(* Logix 5000 project; controller GEA_Test_Chamber vendor 1 type 14 code 196 rev 32.14; software revision 32.04; part 8 of 11 *)
(* tags used below, declared in another part *)
   Heater_Cnt : COUNTER;
   LDO_Error_MSG : INT;
   LDO_LabView_Control : INT;
   LDO_LabView_Control2 : INT;
   LDO_Water_Outlet_Valve : REAL;
   LDO_Water_Outlet_Valve_Flow_SP : REAL;
   LDO_Water_Outlet_Valve_SP : REAL;
   Marcin : BOOL;
   Modbus_LabView_Data : raC_UDT_ModbusServerData;
   nLDO_Rate_REAL : REAL;
   Output_LDO : Output_LDO;

PROGRAM LDO_Chamber   (* main routine LDO_Main *)
VAR
   Act_Time : DINT[7] := ([0] := 2022, [1] := 8, [2] := 30, [4] := 36, [5] := 15, [6] := 396012);
   Actuators_OnOff_Heater : BOOL := 1;
   bPulse05Hz : BOOL := 1;
   bPulse0_1Hz : BOOL := 1;
   bPulse10Hz : BOOL;
   bPulse1Hz : BOOL;
   bPulse1min : BOOL;
   Counter : COUNTER[20] := ([0].PRE := 600, [1].PRE := 1200, [2].PRE := 3300, [3].PRE := 300, [4].PRE := 10, [5].PRE := 14100, [6].PRE := 300, [7].PRE := 2, [8].PRE := 14100, [9].PRE := 300, [10].PRE := 300, [11].PRE := 1500, [12].PRE := 180, [13].PRE := 1620, [14].PRE := 3300, [15].PRE := 300, [16].PRE := 1800, [17].PRE := 1800);
   DRK375_Flow_Change : BOOL;
   DRK375_Flow_InRange : BOOL := 1;
   DRK375_Temp_Change : BOOL;
   DRK375_Temp_InRange : BOOL := 1;
   Flow_Change_Step : INT;
   FVIR_Water_DRK375_Error : REAL := -175.0;
   GasSolenoidOnOff : BOOL := 1;
   Heater_OnOff : BOOL;
   LDO_DRK375_Start : BOOL;
   LDO_LabView_Comm_OK : BOOL;
   LDO_Oil_Step : INT;
   LDO_Step : INT;
   LDO_TestFlow : BOOL;
   LDO_Timer_Delay : TIMER[30] := ([0].PRE := 250, [20].PRE := 30000);
   LDO_Water_DRK375 : REAL := 50.0;
   LDO_Water_float : REAL := 9.0;
   LDO_Water_Flow_DRK375_REG : REAL := -175.0;
   LDO_Water_Flow_DRK375_SP : INT;
   LDO_Water_Outler_Flow : REAL;
   LDO_Water_Outlet : PID := (CTL := 41944064, CA := 1, PE := 1, DVNA := 1, SP := 135.0, KP := 1.0, KI := 0.1, MAXS := 4095.0, SO := 39.631687, MAXO := 50.0, MINO := 25.0, UPD := 0.1, PV := 134.7, ERR := -0.30000305, OUT := 39.631687, PVH := 200.0, DVP := 100.0, MAXI := 4095.0, MAXTIE := 4095.0, DATA[0] := 39.63901, DATA[1] := 52.630035, DATA[2] := 134.7, DATA[3] := -0.30000305, DATA[4] := 135.0, DATA[5] := 0.024420025, DATA[6] := 1.0, DATA[7] := 1.6, DATA[8] := 1.0, DATA[9] := 0.1, DATA[11] := 1.0, DATA[12] := 0.16666667, DATA[16] := 0.024420025);
   LDO_Water_Outlet_2 : PID := (CTL := -2139057280, EN := 1, PE := 1, INI := 1, OLH := 1, DVPA := 1, PVLA := 1, PVHA := 1, SP := 0.5803782, KP := 1.0, KI := 0.1, MAXS := 4095.0, SO := 100.0, MAXO := 100.0, UPD := 0.1, ERR := 0.5803782, OUT := 100.0, MAXI := 4095.0, MAXTIE := 4095.0, DATA[0] := 99.98566, DATA[3] := 0.5803782, DATA[4] := 0.5803782, DATA[5] := 0.024420025, DATA[6] := 1.0, DATA[7] := 1.6, DATA[8] := 1.0, DATA[9] := 0.1, DATA[11] := 1.0, DATA[12] := 0.16666667, DATA[16] := 0.024420025);
   LDO_Water_Outlet_HighLimit : REAL := 140.0;
   LDO_Water_Outlet_LowLimit : REAL := 130.0;
   LDO_Water_Outlet_Temp : REAL := 95.6;
   LDO_Water_Outlet_Valve_PID : REAL;
   LDO_Water_SP_float : REAL := 11.42;
   LDO_Water_Temp_DRK375_SP : INT;
   LDO_Water_Temp_float : REAL := 6.552;
   LDO_Water_Temp_SP_float : REAL := 7.552;
   LDO_WaterHeater_Step : INT := 70;
   Manual : Output_LDO;
   Max_Limit : REAL := 5.88;
   Min_limit : REAL := -4.12;
   New_Time : BOOL := 1;
   Oil_spray_08_ccmin : BOOL;
   Oil_spray_11_ccmin : BOOL;
   Oil_spray_133_ccmin : BOOL;
   ONS : BOOL[32] := ([0] := 1);
   PID_CV : REAL := 100.0;
   PID_puls : BOOL;
   puls_start : BOOL;
   puls_stop : BOOL;
   Pulse : BOOL[32] := ([10] := 1, [12] := 1, [20] := 1);
   Pulses : BOOL[32];
   Reset_Cnt : BOOL;
   Spare_Module : BOOL;
   Start_Test : BOOL;
   Start_Water_Flow : BOOL := 1;
   Step_10_Done : BOOL;
   Step_20_Done : BOOL;
   Step_25_Done : BOOL;
   Step_30_Done : BOOL;
   Step_40_Done : BOOL;
   Step_5_Done : BOOL;
   T_Diff_10 : DINT := 453959;
   T_Diff_20 : DINT := 453659;
   T_Diff_25 : DINT := 405359;
   T_Diff_30 : DINT := 403559;
   T_Diff_40 : DINT := 403379;
   T_Diff_5 : DINT := 455759;
   T_Diff_Step10 : T_DIFF := (T_Diff_sec := 453959);
   T_Diff_Step20 : T_DIFF := (T_Diff_sec := 453659);
   T_Diff_Step25 : T_DIFF := (T_Diff_sec := 405359);
   T_Diff_Step30 : T_DIFF := (T_Diff_sec := 403559);
   T_Diff_Step40 : T_DIFF := (T_Diff_sec := 403379);
   T_Diff_Step5 : T_DIFF := (T_Diff_sec := 455759);
   T_Diff_WaterStep10 : T_DIFF := (T_Diff_sec := 423359);
   T_Diff_WaterStep20 : T_DIFF := (T_Diff_sec := 420059);
   T_Diff_WaterStep40 : T_DIFF := (T_Diff_sec := 405359);
   T_Diff_WaterStep5 : T_DIFF;
   T_Diff_WaterStep50 : T_DIFF := (T_Diff_sec := 391259);
   T_Diff_WaterStep70 : T_DIFF := (T_Diff_sec := 2159);
   T_Diff_WaterStep80 : T_DIFF := (T_Diff_sec := 2459);
   Temp_cal_LDO : DINT := 2425;
   Temp_Change_Step : INT;
   test : BOOL;
   test_Heater_Ready : BOOL := 1;
   Time_Step_10 : DINT[7] := ([0] := 2022, [1] := 8, [2] := 24, [3] := 18, [4] := 30, [5] := 16, [6] := 35);
   Time_Step_20 : DINT[7] := ([0] := 2022, [1] := 8, [2] := 24, [3] := 18, [4] := 35, [5] := 16, [6] := 117);
   Time_Step_25 : DINT[7] := ([0] := 2022, [1] := 8, [2] := 25, [3] := 8, [5] := 16, [6] := 112);
   Time_Step_30 : DINT[7] := ([0] := 2022, [1] := 8, [2] := 25, [3] := 8, [4] := 30, [5] := 16, [6] := 92);
   Time_Step_40 : DINT[7] := ([0] := 2022, [1] := 8, [2] := 25, [3] := 8, [4] := 33, [5] := 16, [6] := 171);
   Time_Step_5 : DINT[7] := ([0] := 2022, [1] := 8, [2] := 24, [3] := 18, [5] := 16, [6] := 621647);
   Timer_Delay : TIMER[30] := ([0].PRE := 100, [0].ACC := 100, [0].EN := 1, [0].DN := 1, [1].PRE := 200, [2].PRE := 500, [3].PRE := 500);
   tof0_1sPulse : TIMER := (PRE := 100, ACC := 100);
   tof10sPulse : TIMER := (PRE := 10000, ACC := 8231, TT := 1, DN := 1);
   tof1sPulse : TIMER := (PRE := 500, ACC := 500);
   tof2sPulse : TIMER := (PRE := 2000, ACC := 236, TT := 1, DN := 1);
   tof30sPulse : TIMER := (PRE := 30000, ACC := 8241, TT := 1, DN := 1);
   ton0_1sPulse : TIMER := (PRE := 100, ACC := 36, EN := 1, TT := 1);
   ton10sPulse : TIMER := (PRE := 10000);
   ton1sPulse : TIMER := (PRE := 500, ACC := 231, EN := 1, TT := 1);
   ton2sPulse : TIMER := (PRE := 2000);
   ton30sPulse : TIMER := (PRE := 30000);
   TON_LifeBit_OFF : TIMER := (PRE := 10000);
   TON_LifeBit_ON : TIMER := (PRE := 10000, ACC := 10000, EN := 1, DN := 1);
   Water_Flow_Calc : REAL := 1084.1355;
   Water_Flow_Calc_float : REAL := 4677.2036;
   Water_Flow_DRK375 : INT := 4677;
   Water_Flow_DRK375_Last : INT := 19;
   Water_Outlet_Calc_LDO : DINT := 1937;
   Water_Outlet_InRange : BOOL;
   Water_Outlet_InRange_LDO : BOOL := 1;
   Water_Outlet_Temp_OK : BOOL;
   Water_Outlet_Valve_LDO : DINT;
   Water_Step_10 : DINT[7] := ([0] := 2022, [1] := 8, [2] := 25, [3] := 3, [5] := 16, [6] := 156);
   Water_Step_10_Done : BOOL;
   Water_Step_20 : DINT[7] := ([0] := 2022, [1] := 8, [2] := 25, [3] := 3, [4] := 55, [5] := 16, [6] := 196);
   Water_Step_20_Done : BOOL;
   Water_Step_40 : DINT;
   Water_Step_401 : DINT[7] := ([0] := 2022, [1] := 8, [2] := 25, [3] := 8, [5] := 16, [6] := 112);
   Water_Step_40_Done : BOOL;
   Water_Step_50 : DINT[7] := ([0] := 2022, [1] := 8, [2] := 25, [3] := 11, [4] := 55, [5] := 16, [6] := 229);
   Water_Step_50_Done : BOOL;
   Water_Step_70 : DINT[7] := ([0] := 2022, [1] := 8, [2] := 30, [5] := 16, [6] := 142);
   Water_Step_70_Done : BOOL;
   Water_Step_80 : DINT[7] := ([0] := 2022, [1] := 8, [2] := 29, [3] := 23, [4] := 55, [5] := 16, [6] := 90);
   Water_Step_80_Done : BOOL;
   Water_T_Diff_10 : DINT := 423359;
   Water_T_Diff_20 : DINT := 420059;
   Water_T_Diff_40 : DINT := 405359;
   Water_T_Diff_50 : DINT := 391259;
   Water_T_Diff_70 : DINT := 2159;
   Water_T_Diff_80 : DINT := 2459;
   Water_Temp_Calc : INT := 289;
   Water_Temp_Calc_float : REAL := 3093.016;
   Water_Temp_DRK375 : INT := 3093;
   Water_Temp_DRK375_Last : REAL := 70.0;
   Water_Time_Step_10 : DINT;
END_VAR

ROUTINE LDO_Control_Valve   (* ladder *)
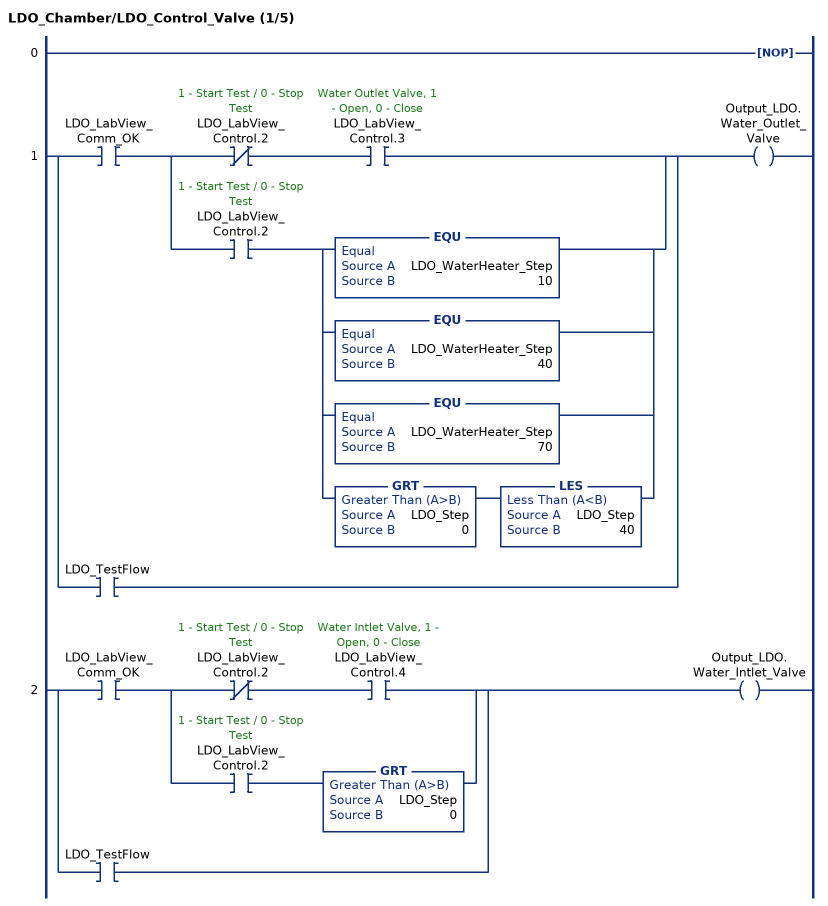
   0: NOP();
   1: [XIC(LDO_LabView_Comm_OK) [XIO(LDO_LabView_Control.2) XIC(LDO_LabView_Control.3) ,XIC(LDO_LabView_Control.2) [EQU(LDO_WaterHeater_Step,10) ,EQU(LDO_WaterHeater_Step,40) ,EQU(LDO_WaterHeater_Step,70) ,GRT(LDO_Step,0) LES(LDO_Step,40) ] ] ,XIC(LDO_TestFlow) ]OTE(Output_LDO.Water_Outlet_Valve);
   2: [XIC(LDO_LabView_Comm_OK) [XIO(LDO_LabView_Control.2) XIC(LDO_LabView_Control.4) ,XIC(LDO_LabView_Control.2) GRT(LDO_Step,0) ] ,XIC(LDO_TestFlow) ]OTE(Output_LDO.Water_Intlet_Valve);
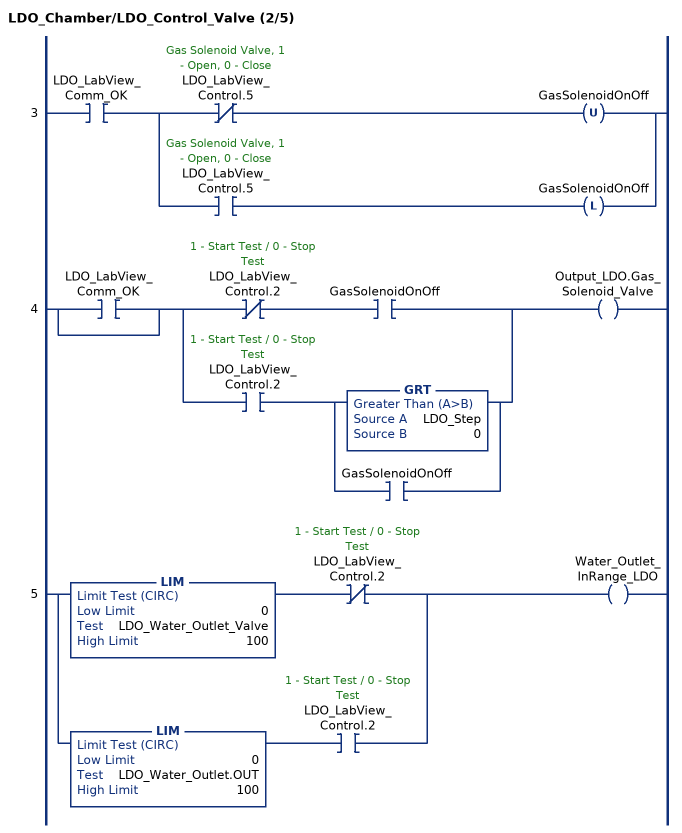
   3: XIC(LDO_LabView_Comm_OK)[XIO(LDO_LabView_Control.5) OTU(GasSolenoidOnOff) ,XIC(LDO_LabView_Control.5) OTL(GasSolenoidOnOff) ];
   4: [XIC(LDO_LabView_Comm_OK) ,][XIO(LDO_LabView_Control.2) XIC(GasSolenoidOnOff) ,XIC(LDO_LabView_Control.2) [GRT(LDO_Step,0) ,XIC(GasSolenoidOnOff) ] ]OTE(Output_LDO.Gas_Solenoid_Valve);
   5: [LIM(0,LDO_Water_Outlet_Valve,100) XIO(LDO_LabView_Control.2) ,LIM(0,LDO_Water_Outlet.OUT,100) XIC(LDO_LabView_Control.2) ]OTE(Water_Outlet_InRange_LDO);
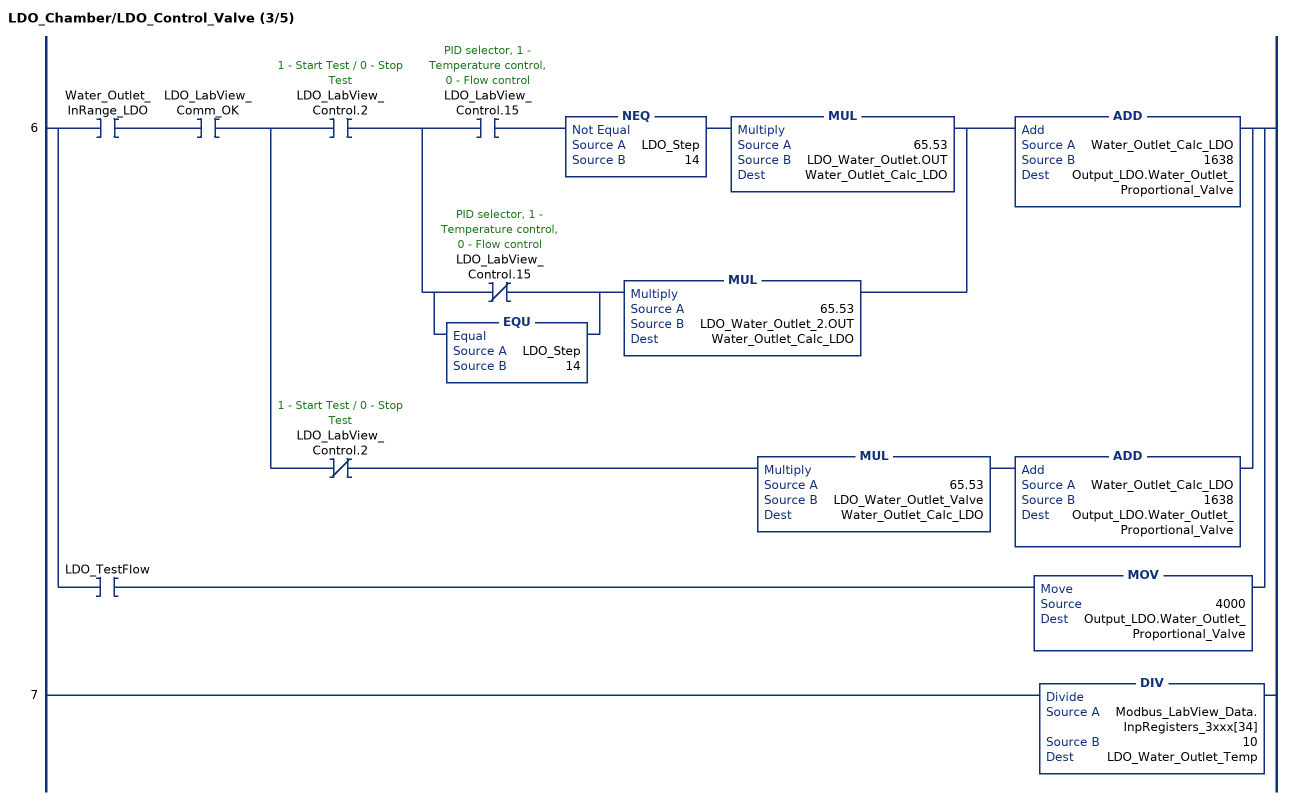
   6: [XIC(Water_Outlet_InRange_LDO) XIC(LDO_LabView_Comm_OK) [XIC(LDO_LabView_Control.2) [XIC(LDO_LabView_Control.15) NEQ(LDO_Step,14) MUL(65.53,LDO_Water_Outlet.OUT,Water_Outlet_Calc_LDO) ,[XIO(LDO_LabView_Control.15) ,EQU(LDO_Step,14) ] MUL(65.53,LDO_Water_Outlet_2.OUT,Water_Outlet_Calc_LDO) ] ADD(Water_Outlet_Calc_LDO,1638,Output_LDO.Water_Outlet_Proportional_Valve) ,XIO(LDO_LabView_Control.2) MUL(65.53,LDO_Water_Outlet_Valve,Water_Outlet_Calc_LDO) ADD(Water_Outlet_Calc_LDO,1638,Output_LDO.Water_Outlet_Proportional_Valve) ] ,XIC(LDO_TestFlow) MOV(4000,Output_LDO.Water_Outlet_Proportional_Valve) ];
   7: DIV(Modbus_LabView_Data.InpRegisters_3xxx[34],10,LDO_Water_Outlet_Temp);
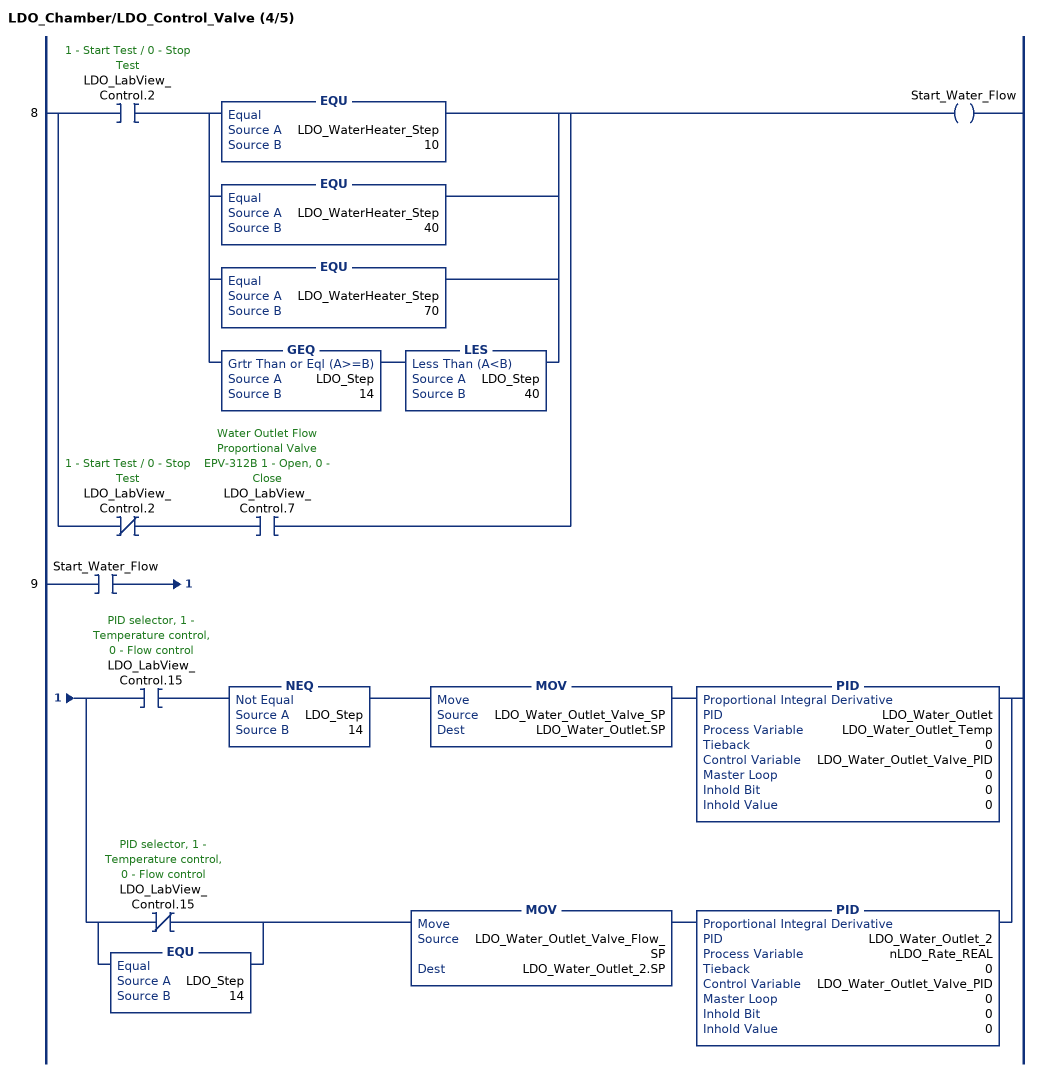
   8: [XIC(LDO_LabView_Control.2) [EQU(LDO_WaterHeater_Step,10) ,EQU(LDO_WaterHeater_Step,40) ,EQU(LDO_WaterHeater_Step,70) ,GEQ(LDO_Step,14) LES(LDO_Step,40) ] ,XIO(LDO_LabView_Control.2) XIC(LDO_LabView_Control.7) ]OTE(Start_Water_Flow);
   9: XIC(Start_Water_Flow)[XIC(LDO_LabView_Control.15) NEQ(LDO_Step,14) MOV(LDO_Water_Outlet_Valve_SP,LDO_Water_Outlet.SP) PID(LDO_Water_Outlet,LDO_Water_Outlet_Temp,0,LDO_Water_Outlet_Valve_PID,0,0,0) ,[XIO(LDO_LabView_Control.15) ,EQU(LDO_Step,14) ] MOV(LDO_Water_Outlet_Valve_Flow_SP,LDO_Water_Outlet_2.SP) PID(LDO_Water_Outlet_2,nLDO_Rate_REAL,0,LDO_Water_Outlet_Valve_PID,0,0,0) ];
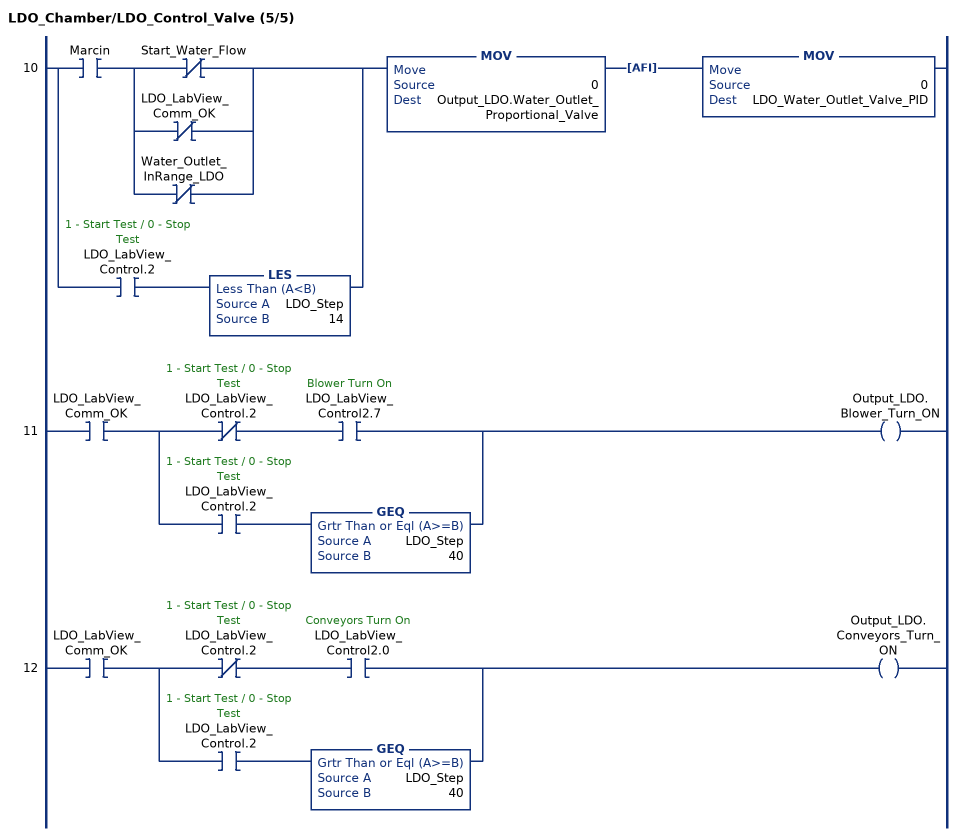
   10: [XIC(Marcin) [XIO(Start_Water_Flow) ,XIO(LDO_LabView_Comm_OK) ,XIO(Water_Outlet_InRange_LDO) ] ,XIC(LDO_LabView_Control.2) LES(LDO_Step,14) ]MOV(0,Output_LDO.Water_Outlet_Proportional_Valve)AFI()MOV(0,LDO_Water_Outlet_Valve_PID);
   11: XIC(LDO_LabView_Comm_OK)[XIO(LDO_LabView_Control.2) XIC(LDO_LabView_Control2.7) ,XIC(LDO_LabView_Control.2) GEQ(LDO_Step,40) ]OTE(Output_LDO.Blower_Turn_ON);
   12: XIC(LDO_LabView_Comm_OK)[XIO(LDO_LabView_Control.2) XIC(LDO_LabView_Control2.0) ,XIC(LDO_LabView_Control.2) GEQ(LDO_Step,40) ]OTE(Output_LDO.Conveyors_Turn_ON);
END_ROUTINE

ROUTINE LDO_Error_MSG   (* ladder *)
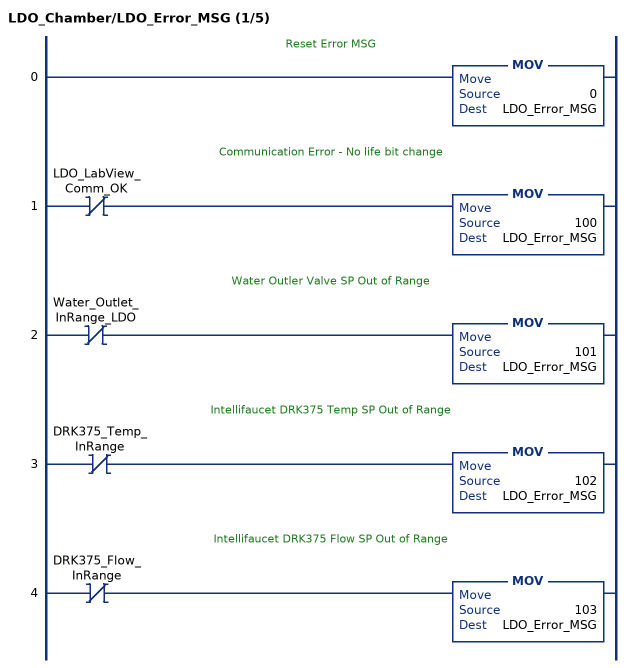
   // Reset Error MSG
   0: MOV(0,LDO_Error_MSG);
   // Communication Error - No life bit change
   1: XIO(LDO_LabView_Comm_OK)MOV(100,LDO_Error_MSG);
   // Water Outler Valve SP Out of Range
   2: XIO(Water_Outlet_InRange_LDO)MOV(101,LDO_Error_MSG);
   // Intellifaucet DRK375 Temp SP Out of Range
   3: XIO(DRK375_Temp_InRange)MOV(102,LDO_Error_MSG);
   // Intellifaucet DRK375 Flow SP Out of Range
   4: XIO(DRK375_Flow_InRange)MOV(103,LDO_Error_MSG);
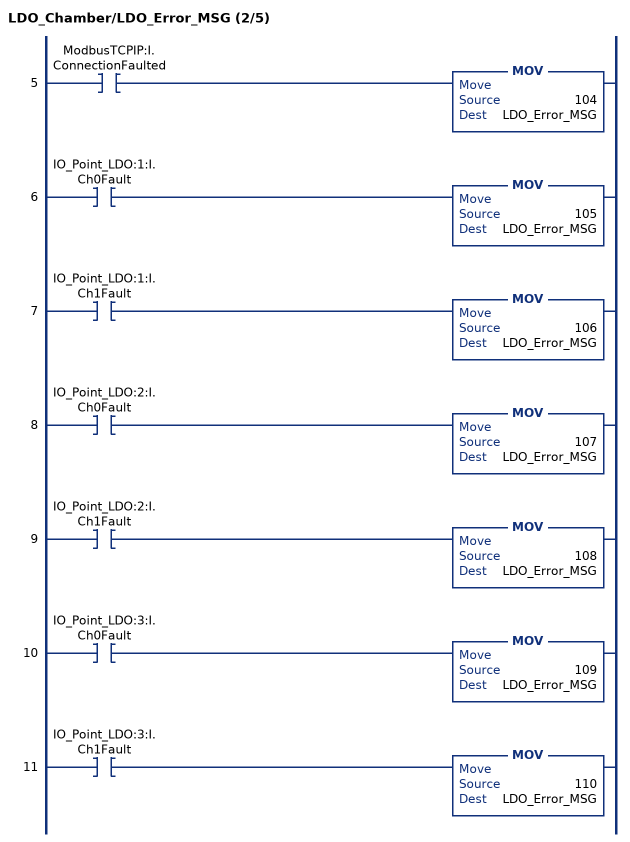
   5: XIC(ModbusTCPIP:I.ConnectionFaulted)MOV(104,LDO_Error_MSG);
   6: XIC(IO_Point_LDO:1:I.Ch0Fault)MOV(105,LDO_Error_MSG);
   7: XIC(IO_Point_LDO:1:I.Ch1Fault)MOV(106,LDO_Error_MSG);
   8: XIC(IO_Point_LDO:2:I.Ch0Fault)MOV(107,LDO_Error_MSG);
   9: XIC(IO_Point_LDO:2:I.Ch1Fault)MOV(108,LDO_Error_MSG);
   10: XIC(IO_Point_LDO:3:I.Ch0Fault)MOV(109,LDO_Error_MSG);
   11: XIC(IO_Point_LDO:3:I.Ch1Fault)MOV(110,LDO_Error_MSG);
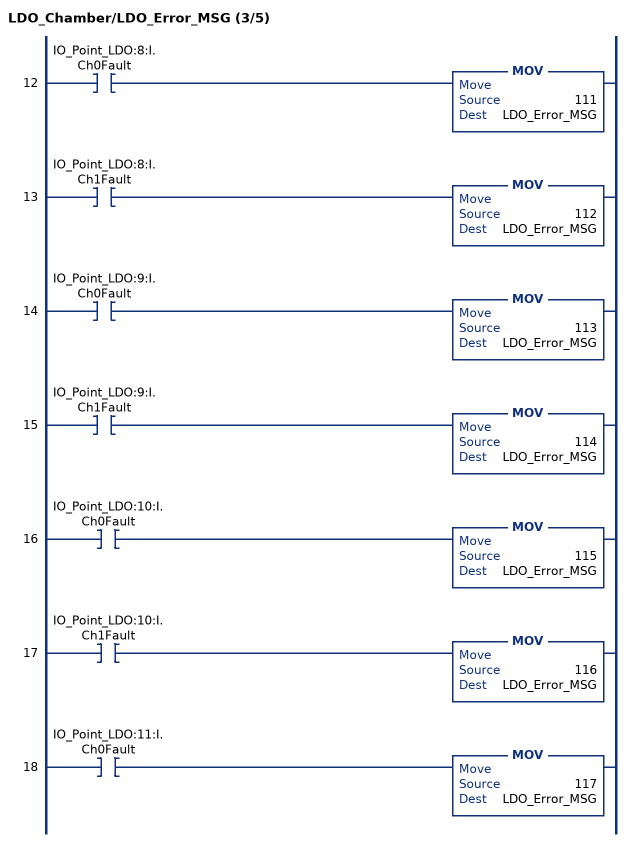
   12: XIC(IO_Point_LDO:8:I.Ch0Fault)MOV(111,LDO_Error_MSG);
   13: XIC(IO_Point_LDO:8:I.Ch1Fault)MOV(112,LDO_Error_MSG);
   14: XIC(IO_Point_LDO:9:I.Ch0Fault)MOV(113,LDO_Error_MSG);
   15: XIC(IO_Point_LDO:9:I.Ch1Fault)MOV(114,LDO_Error_MSG);
   16: XIC(IO_Point_LDO:10:I.Ch0Fault)MOV(115,LDO_Error_MSG);
   17: XIC(IO_Point_LDO:10:I.Ch1Fault)MOV(116,LDO_Error_MSG);
   18: XIC(IO_Point_LDO:11:I.Ch0Fault)MOV(117,LDO_Error_MSG);
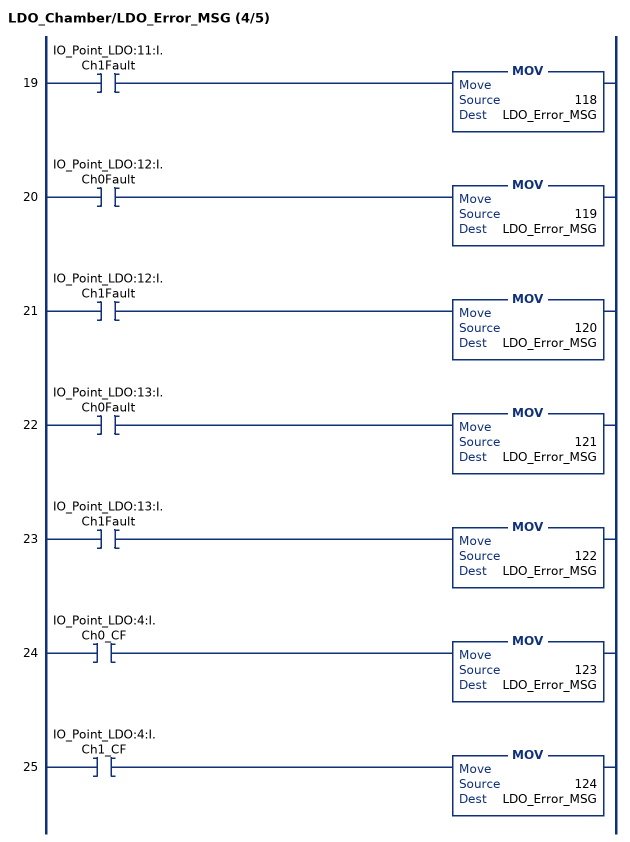
   19: XIC(IO_Point_LDO:11:I.Ch1Fault)MOV(118,LDO_Error_MSG);
   20: XIC(IO_Point_LDO:12:I.Ch0Fault)MOV(119,LDO_Error_MSG);
   21: XIC(IO_Point_LDO:12:I.Ch1Fault)MOV(120,LDO_Error_MSG);
   22: XIC(IO_Point_LDO:13:I.Ch0Fault)MOV(121,LDO_Error_MSG);
   23: XIC(IO_Point_LDO:13:I.Ch1Fault)MOV(122,LDO_Error_MSG);
   24: XIC(IO_Point_LDO:4:I.Ch0_CF)MOV(123,LDO_Error_MSG);
   25: XIC(IO_Point_LDO:4:I.Ch1_CF)MOV(124,LDO_Error_MSG);
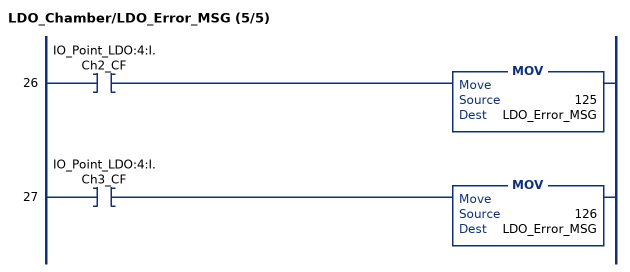
   26: XIC(IO_Point_LDO:4:I.Ch2_CF)MOV(125,LDO_Error_MSG);
   27: XIC(IO_Point_LDO:4:I.Ch3_CF)MOV(126,LDO_Error_MSG);
END_ROUTINE

ROUTINE LDO_Heater_OnOff   (* ladder *)
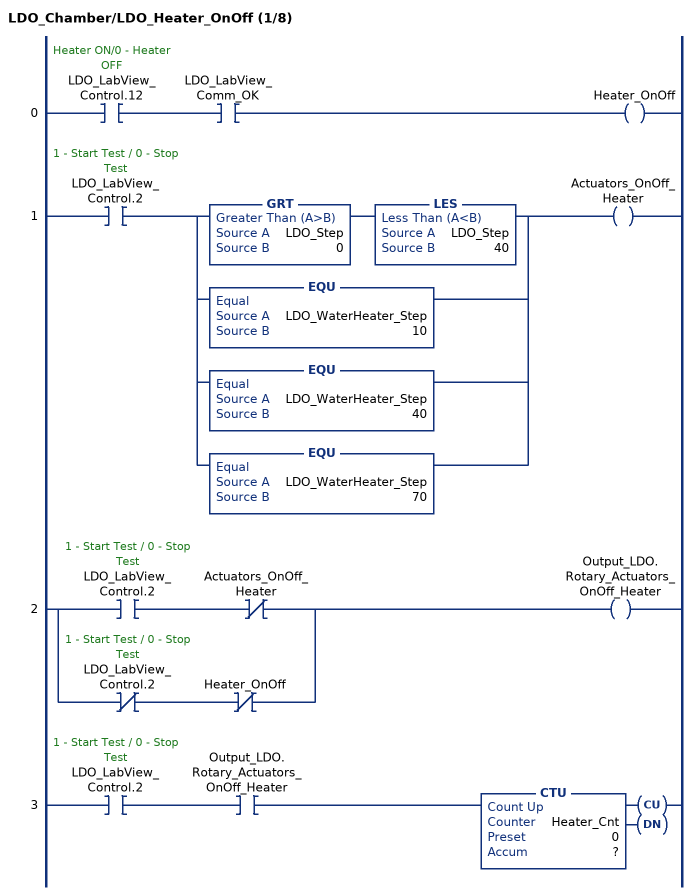
   0: XIC(LDO_LabView_Control.12)XIC(LDO_LabView_Comm_OK)OTE(Heater_OnOff);
   1: XIC(LDO_LabView_Control.2)[GRT(LDO_Step,0) LES(LDO_Step,40) ,EQU(LDO_WaterHeater_Step,10) ,EQU(LDO_WaterHeater_Step,40) ,EQU(LDO_WaterHeater_Step,70) ]OTE(Actuators_OnOff_Heater);
   2: [XIC(LDO_LabView_Control.2) XIO(Actuators_OnOff_Heater) ,XIO(LDO_LabView_Control.2) XIO(Heater_OnOff) ]OTE(Output_LDO.Rotary_Actuators_OnOff_Heater);
   3: XIC(LDO_LabView_Control.2)XIC(Output_LDO.Rotary_Actuators_OnOff_Heater)CTU(Heater_Cnt,?,?);
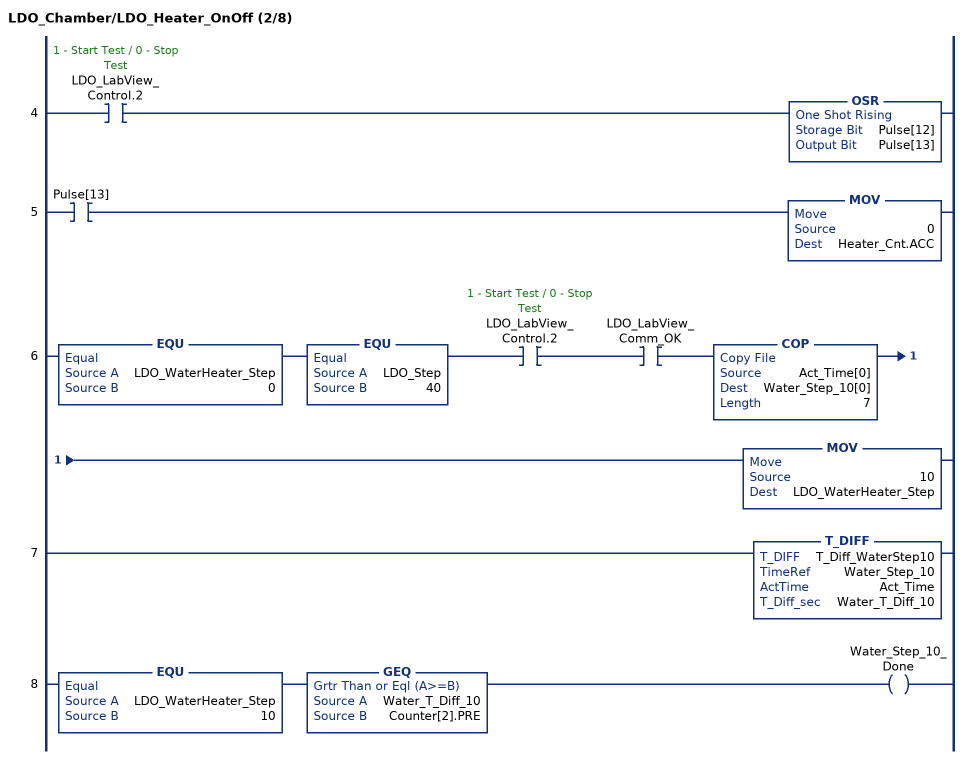
   4: XIC(LDO_LabView_Control.2)OSR(Pulse[12],Pulse[13]);
   5: XIC(Pulse[13])MOV(0,Heater_Cnt.ACC);
   6: EQU(LDO_WaterHeater_Step,0)EQU(LDO_Step,40)XIC(LDO_LabView_Control.2)XIC(LDO_LabView_Comm_OK)COP(Act_Time[0],Water_Step_10[0],7)MOV(10,LDO_WaterHeater_Step);
   7: T_DIFF(T_Diff_WaterStep10,Water_Step_10,Act_Time,Water_T_Diff_10);
   8: EQU(LDO_WaterHeater_Step,10)GEQ(Water_T_Diff_10,Counter[2].PRE)OTE(Water_Step_10_Done);
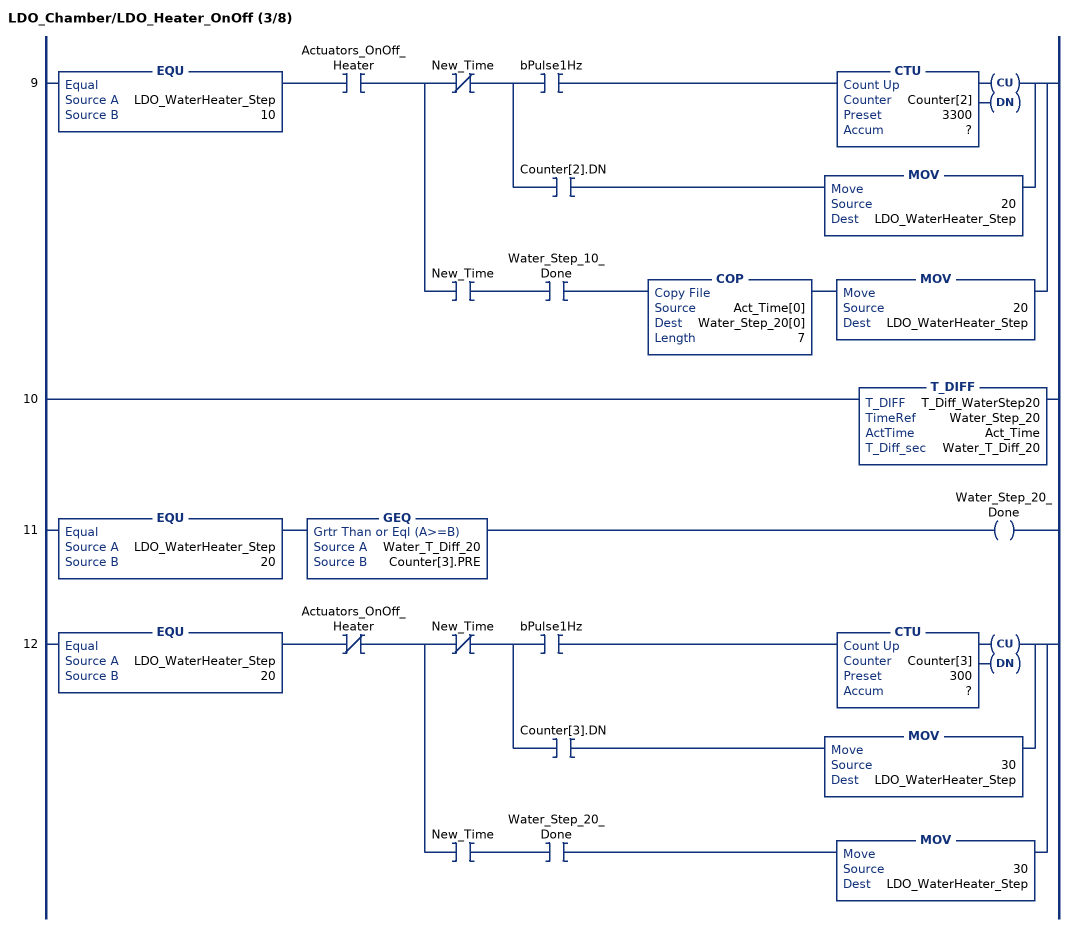
   9: EQU(LDO_WaterHeater_Step,10)XIC(Actuators_OnOff_Heater)[XIO(New_Time) [XIC(bPulse1Hz) CTU(Counter[2],?,?) ,XIC(Counter[2].DN) MOV(20,LDO_WaterHeater_Step) ] ,XIC(New_Time) XIC(Water_Step_10_Done) COP(Act_Time[0],Water_Step_20[0],7) MOV(20,LDO_WaterHeater_Step) ];
   10: T_DIFF(T_Diff_WaterStep20,Water_Step_20,Act_Time,Water_T_Diff_20);
   11: EQU(LDO_WaterHeater_Step,20)GEQ(Water_T_Diff_20,Counter[3].PRE)OTE(Water_Step_20_Done);
   12: EQU(LDO_WaterHeater_Step,20)XIO(Actuators_OnOff_Heater)[XIO(New_Time) [XIC(bPulse1Hz) CTU(Counter[3],?,?) ,XIC(Counter[3].DN) MOV(30,LDO_WaterHeater_Step) ] ,XIC(New_Time) XIC(Water_Step_20_Done) MOV(30,LDO_WaterHeater_Step) ];
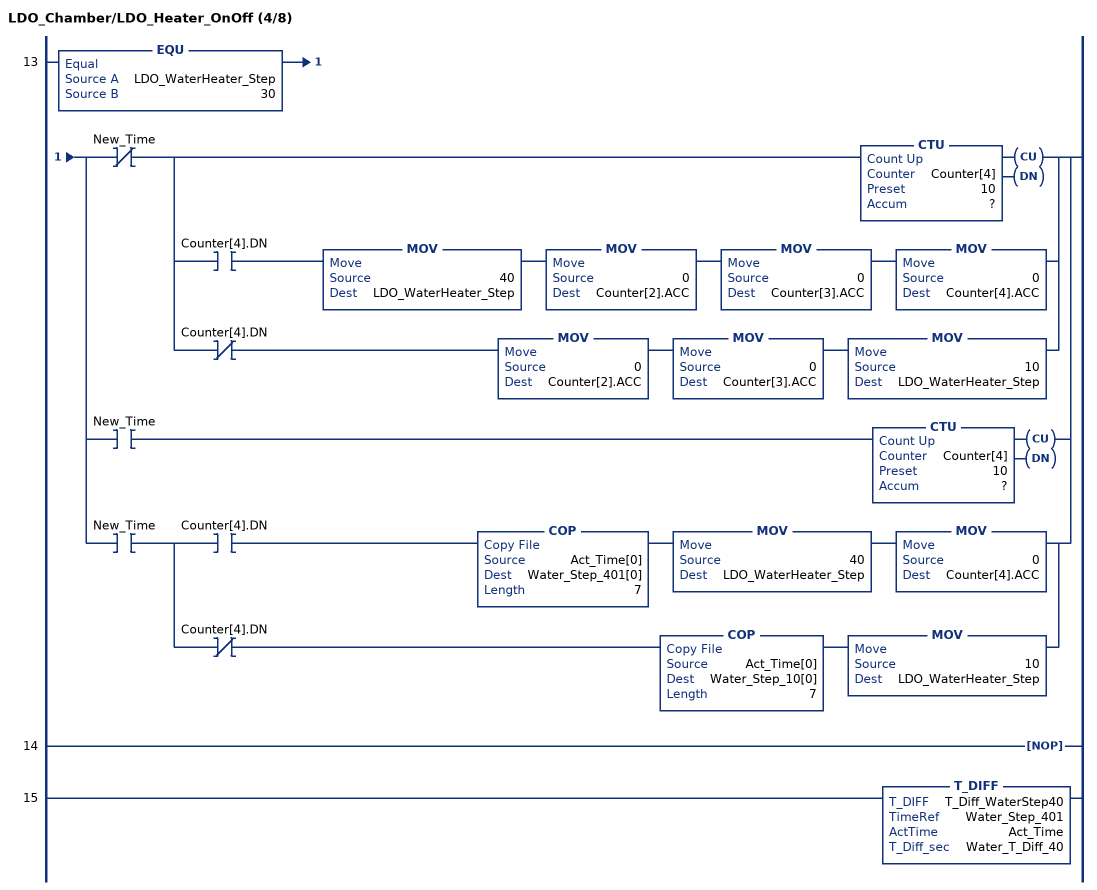
   13: EQU(LDO_WaterHeater_Step,30)[XIO(New_Time) [CTU(Counter[4],?,?) ,XIC(Counter[4].DN) MOV(40,LDO_WaterHeater_Step) MOV(0,Counter[2].ACC) MOV(0,Counter[3].ACC) MOV(0,Counter[4].ACC) ,XIO(Counter[4].DN) MOV(0,Counter[2].ACC) MOV(0,Counter[3].ACC) MOV(10,LDO_WaterHeater_Step) ] ,XIC(New_Time) CTU(Counter[4],?,?) ,XIC(New_Time) [XIC(Counter[4].DN) COP(Act_Time[0],Water_Step_401[0],7) MOV(40,LDO_WaterHeater_Step) MOV(0,Counter[4].ACC) ,XIO(Counter[4].DN) COP(Act_Time[0],Water_Step_10[0],7) MOV(10,LDO_WaterHeater_Step) ] ];
   14: NOP();
   15: T_DIFF(T_Diff_WaterStep40,Water_Step_401,Act_Time,Water_T_Diff_40);
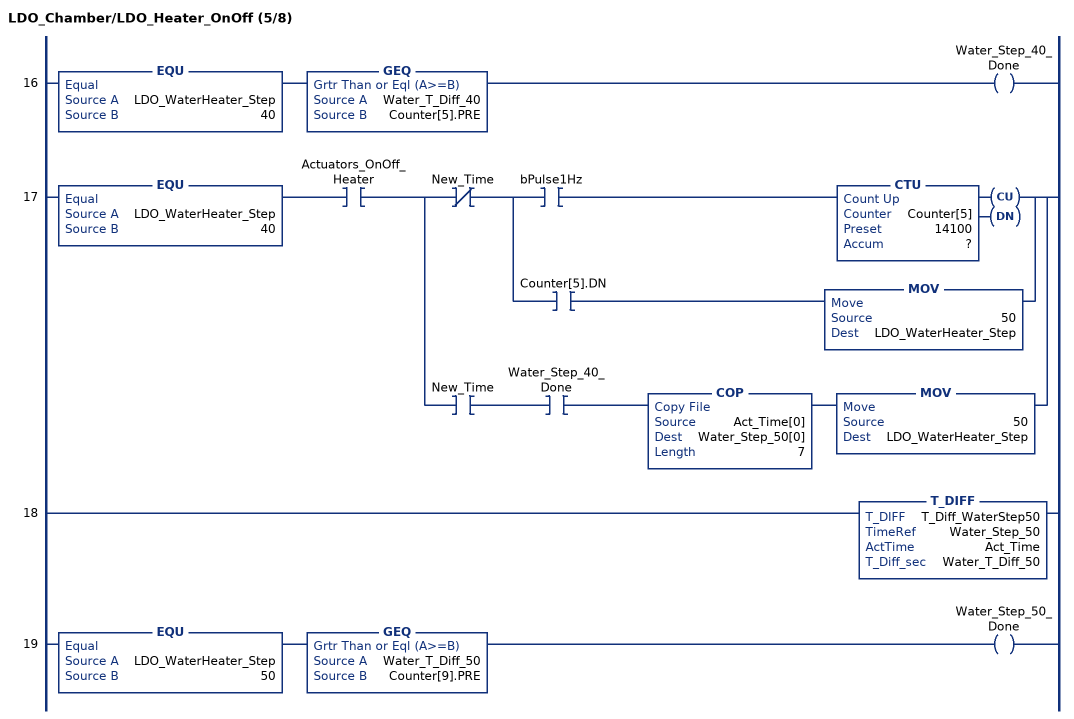
   16: EQU(LDO_WaterHeater_Step,40)GEQ(Water_T_Diff_40,Counter[5].PRE)OTE(Water_Step_40_Done);
   17: EQU(LDO_WaterHeater_Step,40)XIC(Actuators_OnOff_Heater)[XIO(New_Time) [XIC(bPulse1Hz) CTU(Counter[5],?,?) ,XIC(Counter[5].DN) MOV(50,LDO_WaterHeater_Step) ] ,XIC(New_Time) XIC(Water_Step_40_Done) COP(Act_Time[0],Water_Step_50[0],7) MOV(50,LDO_WaterHeater_Step) ];
   18: T_DIFF(T_Diff_WaterStep50,Water_Step_50,Act_Time,Water_T_Diff_50);
   19: EQU(LDO_WaterHeater_Step,50)GEQ(Water_T_Diff_50,Counter[9].PRE)OTE(Water_Step_50_Done);
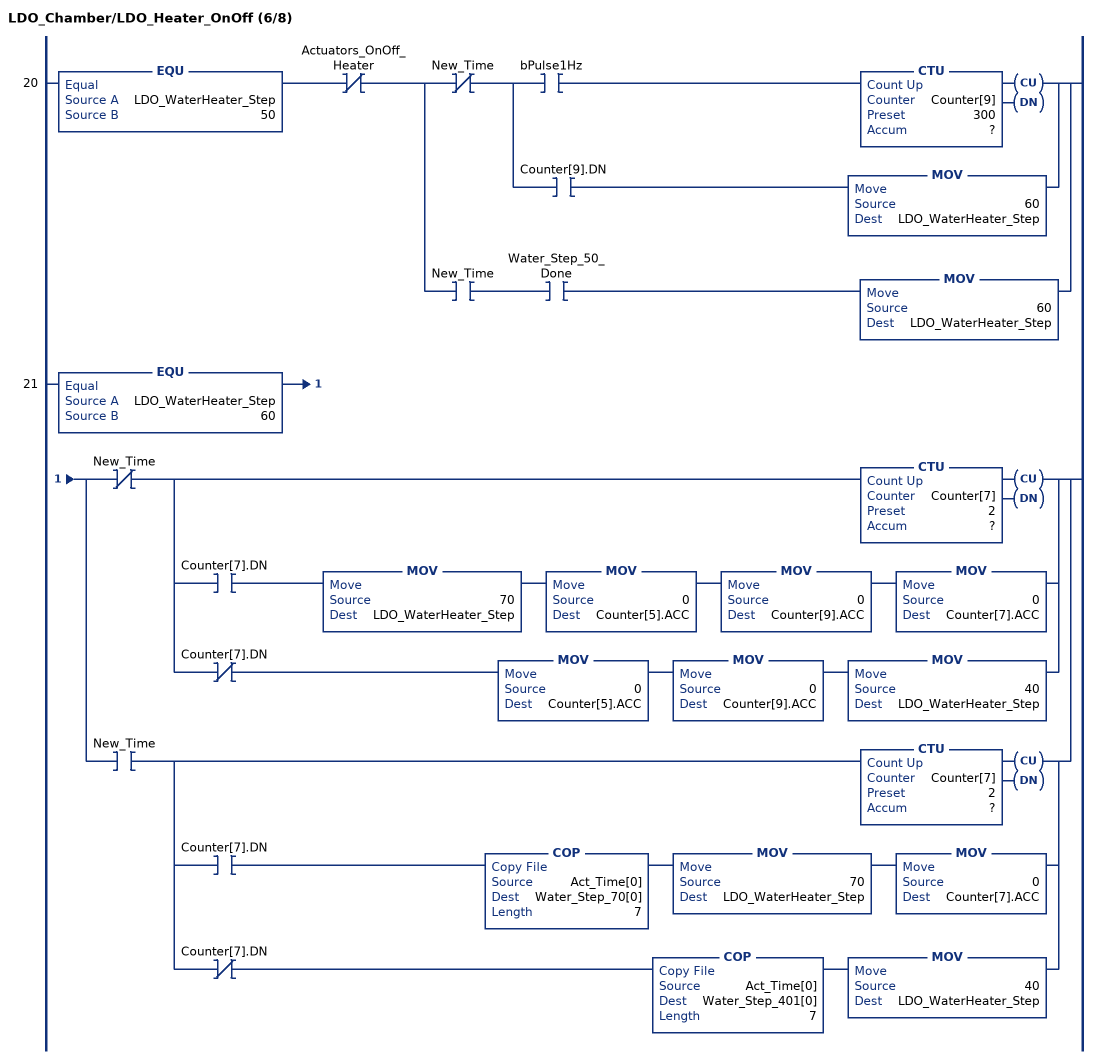
   20: EQU(LDO_WaterHeater_Step,50)XIO(Actuators_OnOff_Heater)[XIO(New_Time) [XIC(bPulse1Hz) CTU(Counter[9],?,?) ,XIC(Counter[9].DN) MOV(60,LDO_WaterHeater_Step) ] ,XIC(New_Time) XIC(Water_Step_50_Done) MOV(60,LDO_WaterHeater_Step) ];
   21: EQU(LDO_WaterHeater_Step,60)[XIO(New_Time) [CTU(Counter[7],?,?) ,XIC(Counter[7].DN) MOV(70,LDO_WaterHeater_Step) MOV(0,Counter[5].ACC) MOV(0,Counter[9].ACC) MOV(0,Counter[7].ACC) ,XIO(Counter[7].DN) MOV(0,Counter[5].ACC) MOV(0,Counter[9].ACC) MOV(40,LDO_WaterHeater_Step) ] ,XIC(New_Time) [CTU(Counter[7],?,?) ,XIC(Counter[7].DN) COP(Act_Time[0],Water_Step_70[0],7) MOV(70,LDO_WaterHeater_Step) MOV(0,Counter[7].ACC) ,XIO(Counter[7].DN) COP(Act_Time[0],Water_Step_401[0],7) MOV(40,LDO_WaterHeater_Step) ] ];
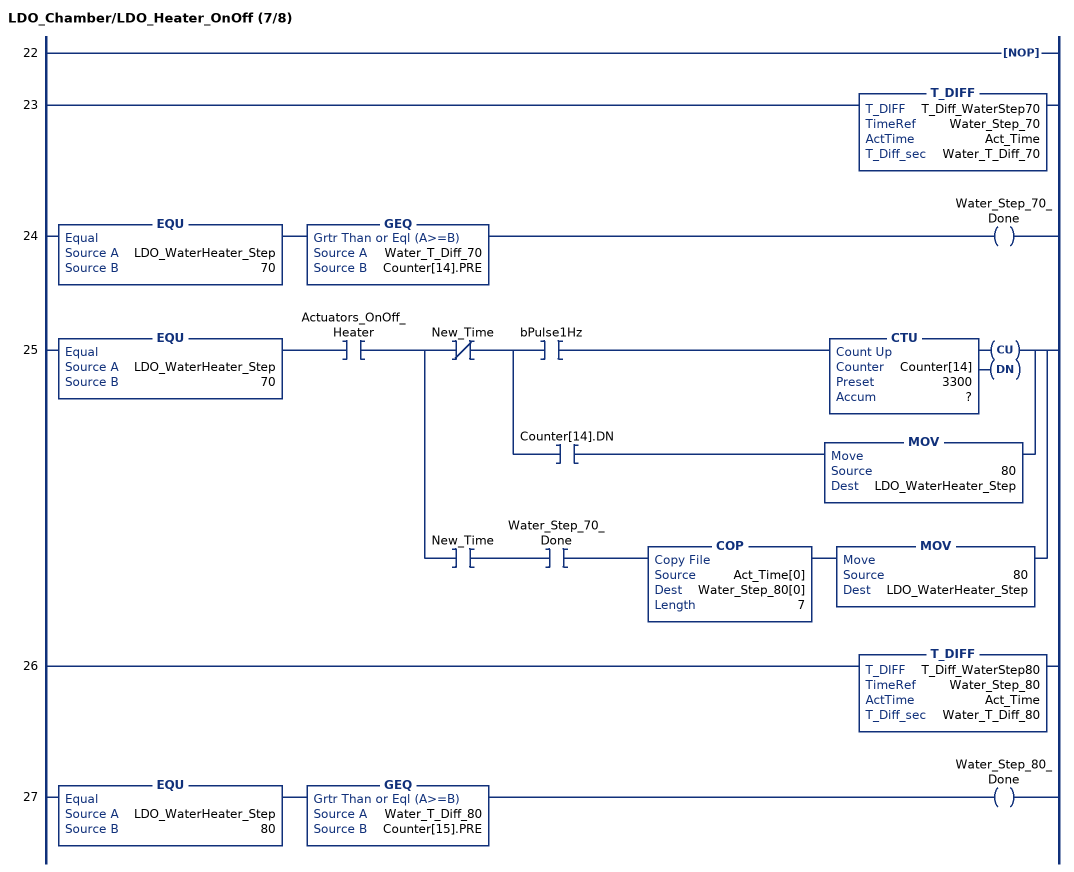
   22: NOP();
   23: T_DIFF(T_Diff_WaterStep70,Water_Step_70,Act_Time,Water_T_Diff_70);
   24: EQU(LDO_WaterHeater_Step,70)GEQ(Water_T_Diff_70,Counter[14].PRE)OTE(Water_Step_70_Done);
   25: EQU(LDO_WaterHeater_Step,70)XIC(Actuators_OnOff_Heater)[XIO(New_Time) [XIC(bPulse1Hz) CTU(Counter[14],?,?) ,XIC(Counter[14].DN) MOV(80,LDO_WaterHeater_Step) ] ,XIC(New_Time) XIC(Water_Step_70_Done) COP(Act_Time[0],Water_Step_80[0],7) MOV(80,LDO_WaterHeater_Step) ];
   26: T_DIFF(T_Diff_WaterStep80,Water_Step_80,Act_Time,Water_T_Diff_80);
   27: EQU(LDO_WaterHeater_Step,80)GEQ(Water_T_Diff_80,Counter[15].PRE)OTE(Water_Step_80_Done);
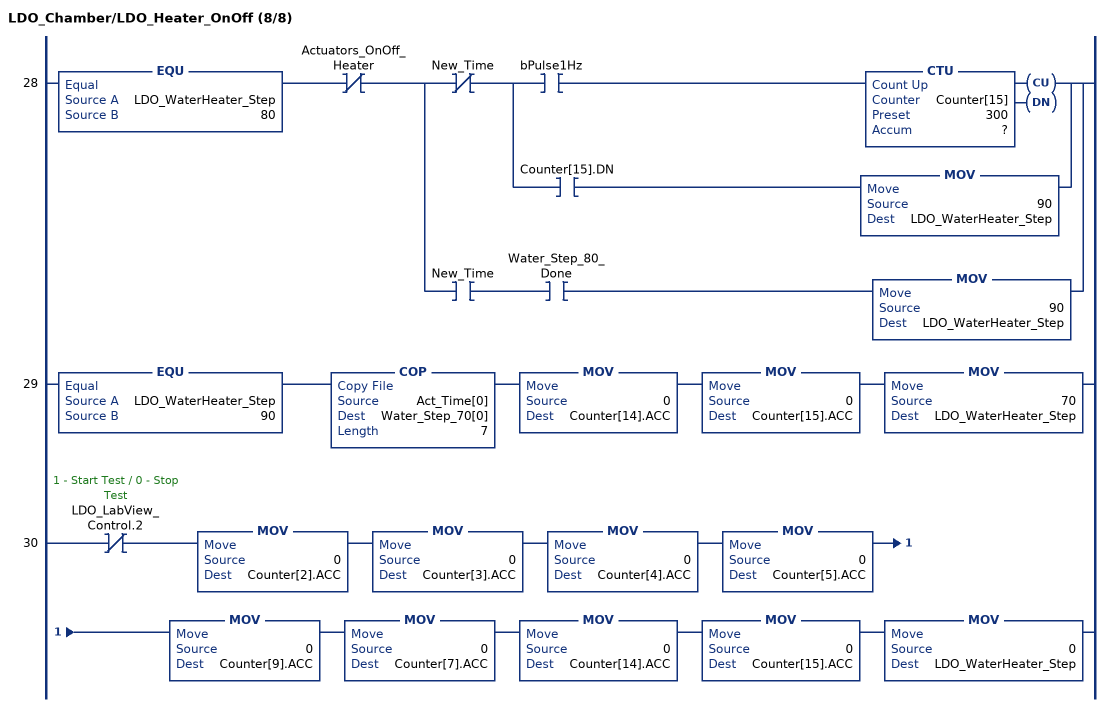
   28: EQU(LDO_WaterHeater_Step,80)XIO(Actuators_OnOff_Heater)[XIO(New_Time) [XIC(bPulse1Hz) CTU(Counter[15],?,?) ,XIC(Counter[15].DN) MOV(90,LDO_WaterHeater_Step) ] ,XIC(New_Time) XIC(Water_Step_80_Done) MOV(90,LDO_WaterHeater_Step) ];
   29: EQU(LDO_WaterHeater_Step,90)COP(Act_Time[0],Water_Step_70[0],7)MOV(0,Counter[14].ACC)MOV(0,Counter[15].ACC)MOV(70,LDO_WaterHeater_Step);
   30: XIO(LDO_LabView_Control.2)MOV(0,Counter[2].ACC)MOV(0,Counter[3].ACC)MOV(0,Counter[4].ACC)MOV(0,Counter[5].ACC)MOV(0,Counter[9].ACC)MOV(0,Counter[7].ACC)MOV(0,Counter[14].ACC)MOV(0,Counter[15].ACC)MOV(0,LDO_WaterHeater_Step);
END_ROUTINE
